// LS Electric XG5000 project: T7_ETH_485_20201209_AfterHeat_Edit
// PLC NewPLC
// module base 0 slot 1: 내장위치결정:XBF-PO02E (오픈컬렉터형, 2축)
// module base 0 slot 2: Cnet:XBL-C41A (Cnet 통신 모듈(RS-422/485))

PROGRAM 7k_pwm (task: 스캔 프로그램)

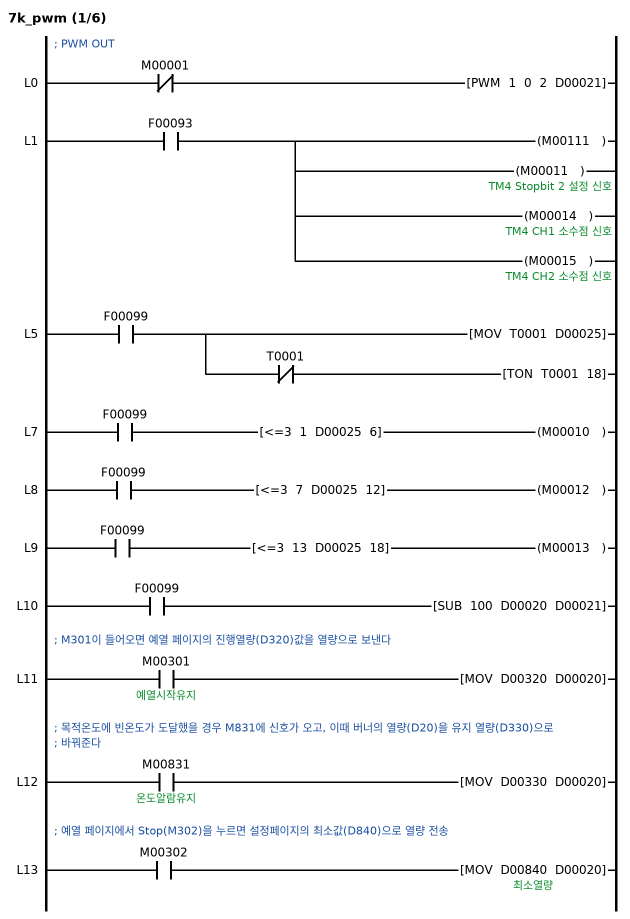
; L0
LOAD NOT  M00001
PWM       1 0 2 D00021
// output comment: PWM OUT
; L1
LOAD      F00093
OUT       M00111
OUT       M00011	// TM4 Stopbit 2 설정 신호
OUT       M00014	// TM4 CH1 소수점 신호
OUT       M00015	// TM4 CH2 소수점 신호
; L5
LOAD      F00099
MOV       T0001 D00025
AND NOT   T0001
TON       T0001 18
; L7
LOAD      F00099
AND<=3    1 D00025 6
OUT       M00010
; L8
LOAD      F00099
AND<=3    7 D00025 12
OUT       M00012
; L9
LOAD      F00099
AND<=3    13 D00025 18
OUT       M00013
; L10
LOAD      F00099
SUB       100 D00020 D00021
; L11
LOAD      M00301	// 예열시작유지
MOV       D00320 D00020
// output comment: M301이 들어오면 예열 페이지의 진행열량(D320)값을 열량으로 보낸다
; L12
LOAD      M00831	// 온도알람유지
MOV       D00330 D00020
// output comment: 목적온도에 빈온도가 도달했을 경우 M831에 신호가 오고, 이때 버너의 열량(D20)을 유지 열량(D330)으로 바꿔준다
; L13
LOAD      M00302
MOV       D00840 D00020	// 최소열량
// output comment: 예열 페이지에서 Stop(M302)을 누르면 설정페이지의 최소값(D840)으로 열량 전송

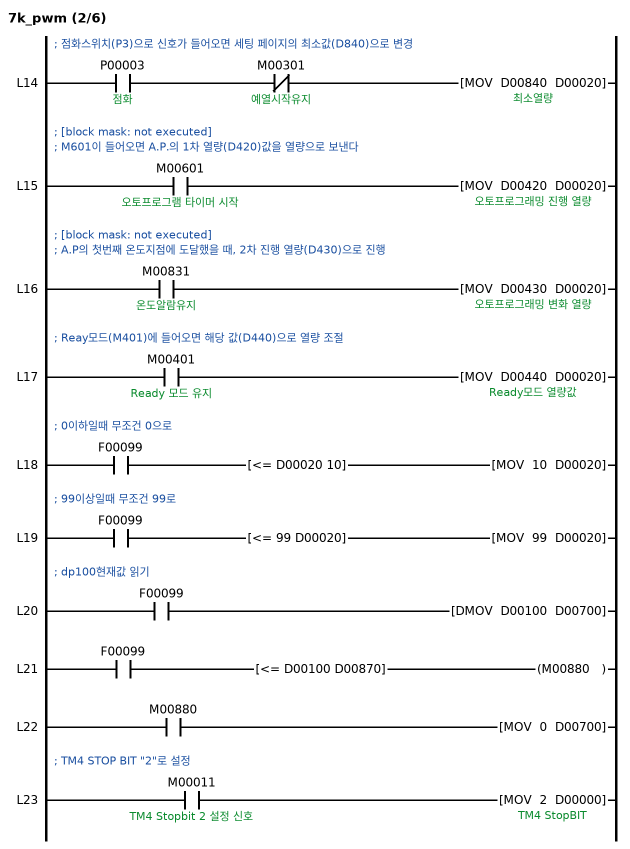
; L14
LOAD      P00003	// 점화
AND NOT   M00301	// 예열시작유지
MOV       D00840 D00020	// 최소열량
// output comment: 점화스위치(P3)으로 신호가 들어오면 세팅 페이지의 최소값(D840)으로 변경
; L15 (block mask: not executed)
LOAD      M00601	// 오토프로그램 타이머 시작
MOV       D00420 D00020	// 오토프로그래밍 진행 열량
// output comment: M601이 들어오면 A.P.의 1차 열량(D420)값을 열량으로 보낸다
; L16 (block mask: not executed)
LOAD      M00831	// 온도알람유지
MOV       D00430 D00020	// 오토프로그래밍 변화 열량
// output comment: A.P의 첫번째 온도지점에 도달했을 때, 2차 진행 열량(D430)으로 진행
; L17
LOAD      M00401	// Ready 모드 유지
MOV       D00440 D00020	// Ready모드 열량값
// output comment: Reay모드(M401)에 들어오면 해당 값(D440)으로 열량 조절
; L18
LOAD      F00099
AND<=     D00020 10
MOV       10 D00020
// output comment: 0이하일때 무조건 0으로
; L19
LOAD      F00099
AND<=     99 D00020
MOV       99 D00020
// output comment: 99이상일때 무조건 99로
; L20
LOAD      F00099
DMOV      D00100 D00700
// output comment: dp100현재값 읽기
; L21
LOAD      F00099
AND<=     D00100 D00870
OUT       M00880
; L22
LOAD      M00880
MOV       0 D00700
; L23
LOAD      M00011	// TM4 Stopbit 2 설정 신호
MOV       2 D00000	// TM4 StopBIT
// output comment: TM4 STOP BIT "2"로 설정

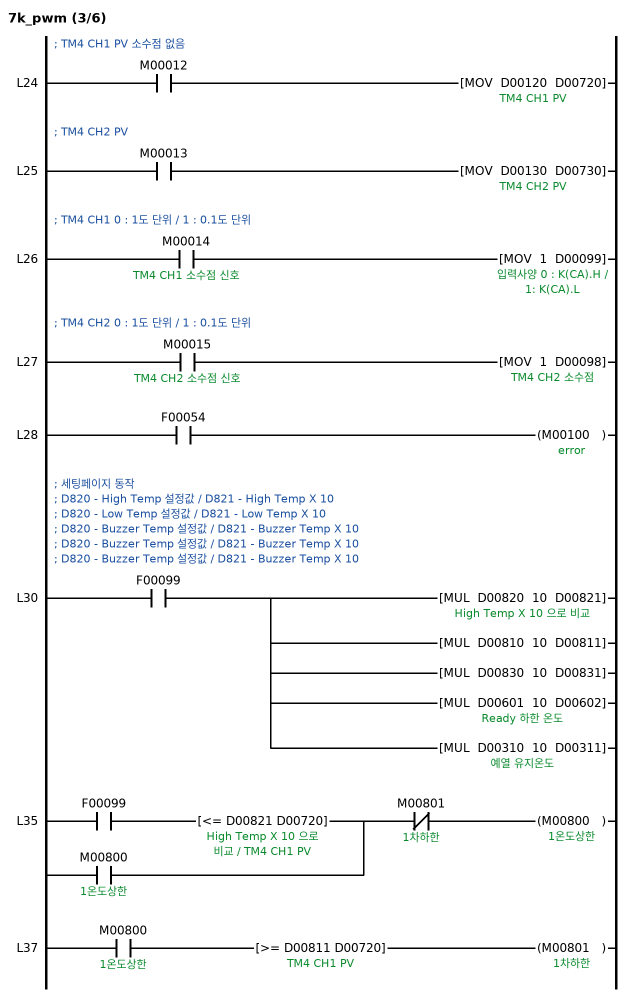
; L24
LOAD      M00012
MOV       D00120 D00720	// TM4 CH1 PV
// output comment: TM4 CH1 PV 소수점 없음
; L25
LOAD      M00013
MOV       D00130 D00730	// TM4 CH2 PV
// output comment: TM4 CH2 PV
; L26
LOAD      M00014	// TM4 CH1 소수점 신호
MOV       1 D00099	// 입력사양 0 : K(CA).H / 1: K(CA).L
// output comment: TM4 CH1 0 : 1도 단위 / 1 : 0.1도 단위
; L27
LOAD      M00015	// TM4 CH2 소수점 신호
MOV       1 D00098	// TM4 CH2 소수점
// output comment: TM4 CH2 0 : 1도 단위 / 1 : 0.1도 단위
; L28
LOAD      F00054
OUT       M00100	// error
// 세팅페이지 동작
; L30
LOAD      F00099
MUL       D00820 10 D00821	// High Temp X 10 으로 비교
MUL       D00810 10 D00811
MUL       D00830 10 D00831
MUL       D00601 10 D00602	// Ready 하한 온도
MUL       D00310 10 D00311	// 예열 유지온도
// output comment: D820 - High Temp 설정값 / D821 - High Temp X 10
// output comment: D820 - Low Temp 설정값 / D821 - Low Temp X 10
// output comment: D820 - Buzzer Temp 설정값 / D821 - Buzzer Temp X 10
// output comment: D820 - Buzzer Temp 설정값 / D821 - Buzzer Temp X 10
// output comment: D820 - Buzzer Temp 설정값 / D821 - Buzzer Temp X 10
; L35
LOAD      F00099
AND<=     D00821 D00720	// High Temp X 10 으로 비교 / TM4 CH1 PV
OR        M00800	// 1온도상한
AND NOT   M00801	// 1차하한
OUT       M00800	// 1온도상한
; L37
LOAD      M00800	// 1온도상한
AND>=     D00811 D00720	// TM4 CH1 PV
OUT       M00801	// 1차하한

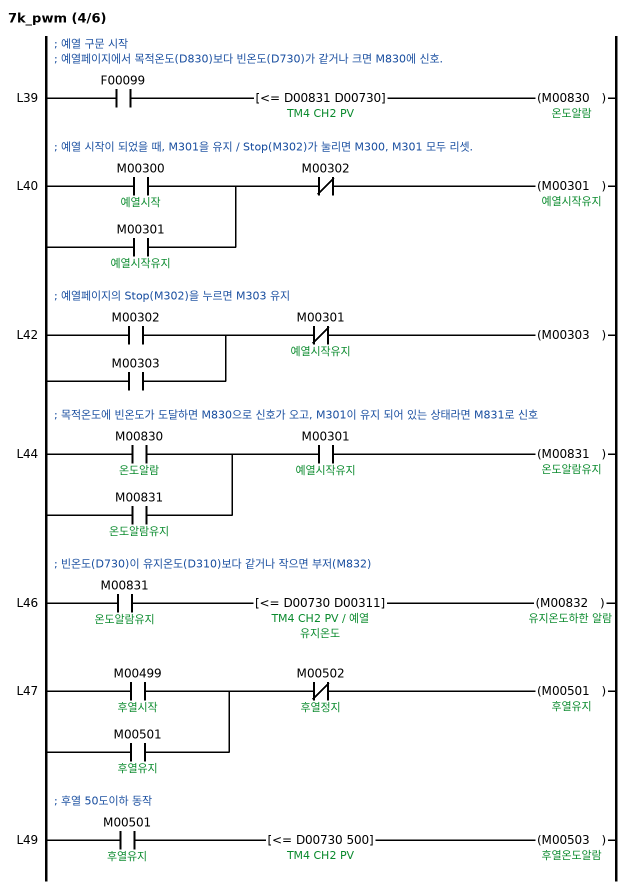
// 예열 구문 시작
; L39
LOAD      F00099
AND<=     D00831 D00730	// TM4 CH2 PV
OUT       M00830	// 온도알람
// output comment: 예열페이지에서 목적온도(D830)보다 빈온도(D730)가 같거나 크면 M830에 신호.
; L40
LOAD      M00300	// 예열시작
OR        M00301	// 예열시작유지
AND NOT   M00302
OUT       M00301	// 예열시작유지
// output comment: 예열 시작이 되었을 때, M301을 유지 / Stop(M302)가 눌리면 M300, M301 모두 리셋.
; L42
LOAD      M00302
OR        M00303
AND NOT   M00301	// 예열시작유지
OUT       M00303
// output comment: 예열페이지의 Stop(M302)을 누르면 M303 유지
; L44
LOAD      M00830	// 온도알람
OR        M00831	// 온도알람유지
AND       M00301	// 예열시작유지
OUT       M00831	// 온도알람유지
// output comment: 목적온도에 빈온도가 도달하면 M830으로 신호가 오고, M301이 유지 되어 있는 상태라면 M831로 신호
; L46
LOAD      M00831	// 온도알람유지
AND<=     D00730 D00311	// TM4 CH2 PV / 예열 유지온도
OUT       M00832	// 유지온도하한 알람
// output comment: 빈온도(D730)이 유지온도(D310)보다 같거나 작으면 부저(M832)
; L47
LOAD      M00499	// 후열시작
OR        M00501	// 후열유지
AND NOT   M00502	// 후열정지
OUT       M00501	// 후열유지
; L49
LOAD      M00501	// 후열유지
AND<=     D00730 500	// TM4 CH2 PV
OUT       M00503	// 후열온도알람
// output comment: 후열 50도이하 동작

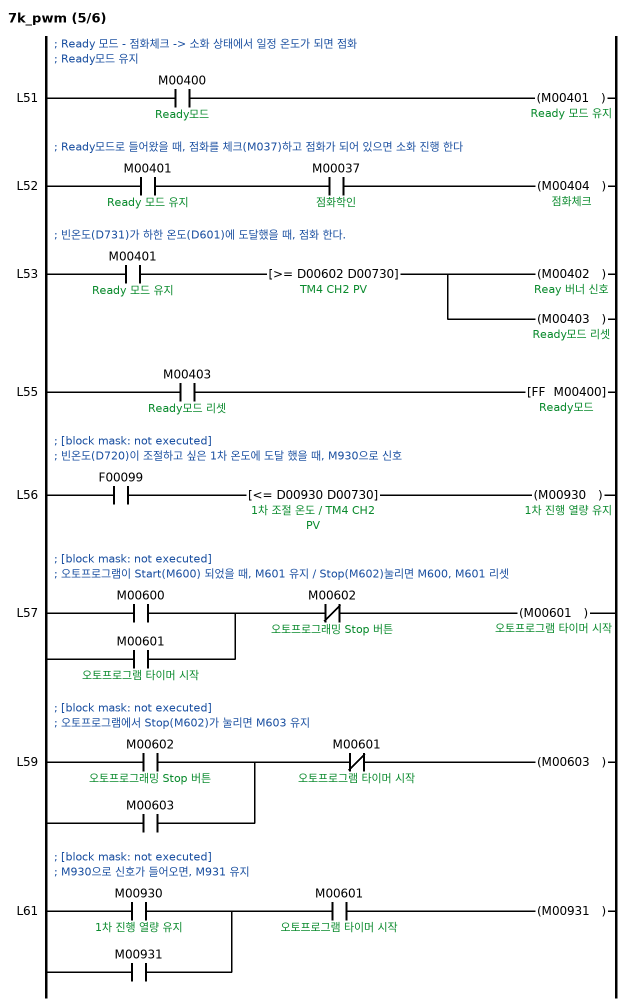
// Ready 모드 - 점화체크 -> 소화 상태에서 일정 온도가 되면 점화
; L51
LOAD      M00400	// Ready모드
OUT       M00401	// Ready 모드 유지
// output comment: Ready모드 유지
; L52
LOAD      M00401	// Ready 모드 유지
AND       M00037	// 점화학인
OUT       M00404	// 점화체크
// output comment: Ready모드로 들어왔을 때, 점화를 체크(M037)하고 점화가 되어 있으면 소화 진행 한다
; L53
LOAD      M00401	// Ready 모드 유지
AND>=     D00602 D00730	// TM4 CH2 PV
OUT       M00402	// Reay 버너 신호
OUT       M00403	// Ready모드 리셋
// output comment: 빈온도(D731)가 하한 온도(D601)에 도달했을 때, 점화 한다.
; L55
LOAD      M00403	// Ready모드 리셋
FF        M00400	// Ready모드
; L56 (block mask: not executed)
LOAD      F00099
AND<=     D00930 D00730	// 1차 조절 온도 / TM4 CH2 PV
OUT       M00930	// 1차 진행 열량 유지
// output comment: 빈온도(D720)이 조절하고 싶은 1차 온도에 도달 했을 때, M930으로 신호
; L57 (block mask: not executed)
LOAD      M00600
OR        M00601	// 오토프로그램 타이머 시작
AND NOT   M00602	// 오토프로그래밍 Stop 버튼
OUT       M00601	// 오토프로그램 타이머 시작
// output comment: 오토프로그램이 Start(M600) 되었을 때, M601 유지 / Stop(M602)눌리면 M600, M601 리셋
; L59 (block mask: not executed)
LOAD      M00602	// 오토프로그래밍 Stop 버튼
OR        M00603
AND NOT   M00601	// 오토프로그램 타이머 시작
OUT       M00603
// output comment: 오토프로그램에서 Stop(M602)가 눌리면 M603 유지
; L61 (block mask: not executed)
LOAD      M00930	// 1차 진행 열량 유지
OR        M00931
AND       M00601	// 오토프로그램 타이머 시작
OUT       M00931
// output comment: M930으로 신호가 들어오면, M931 유지

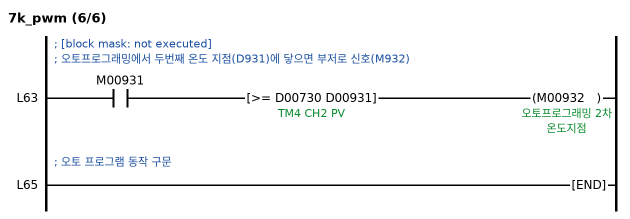
; L63 (block mask: not executed)
LOAD      M00931
AND>=     D00730 D00931	// TM4 CH2 PV
OUT       M00932	// 오토프로그래밍 2차 온도지점
// output comment: 오토프로그래밍에서 두번째 온도 지점(D931)에 닿으면 부저로 신호(M932)
// 오토 프로그램 동작 구문
; L65
END

PROGRAM 타이머 (task: 스캔 프로그램)

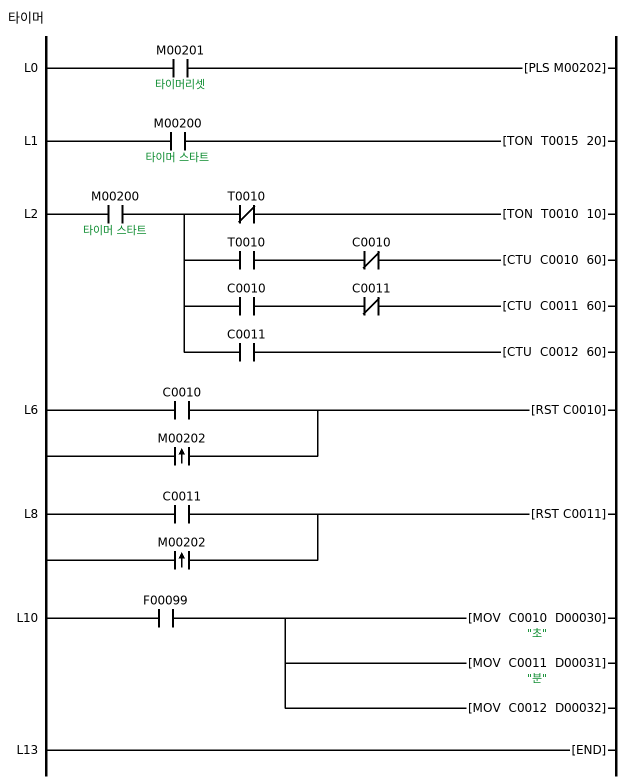
; L0
LOAD      M00201	// 타이머리셋
OUTP      M00202
; L1
LOAD      M00200	// 타이머 스타트
TON       T0015 20
; L2
LOAD      M00200	// 타이머 스타트
MPUSH
AND NOT   T0010
TON       T0010 10
MLOAD
AND       T0010
AND NOT   C0010
CTU       C0010 60
MLOAD
AND       C0010
AND NOT   C0011
CTU       C0011 60
MPOP
AND       C0011
CTU       C0012 60
; L6
LOAD      C0010
ORP       M00202
RST       C0010
; L8
LOAD      C0011
ORP       M00202
RST       C0011
; L10
LOAD      F00099
MOV       C0010 D00030	// "초"
MOV       C0011 D00031	// "분"
MOV       C0012 D00032
; L13
END

PROGRAM control (task: 스캔 프로그램)

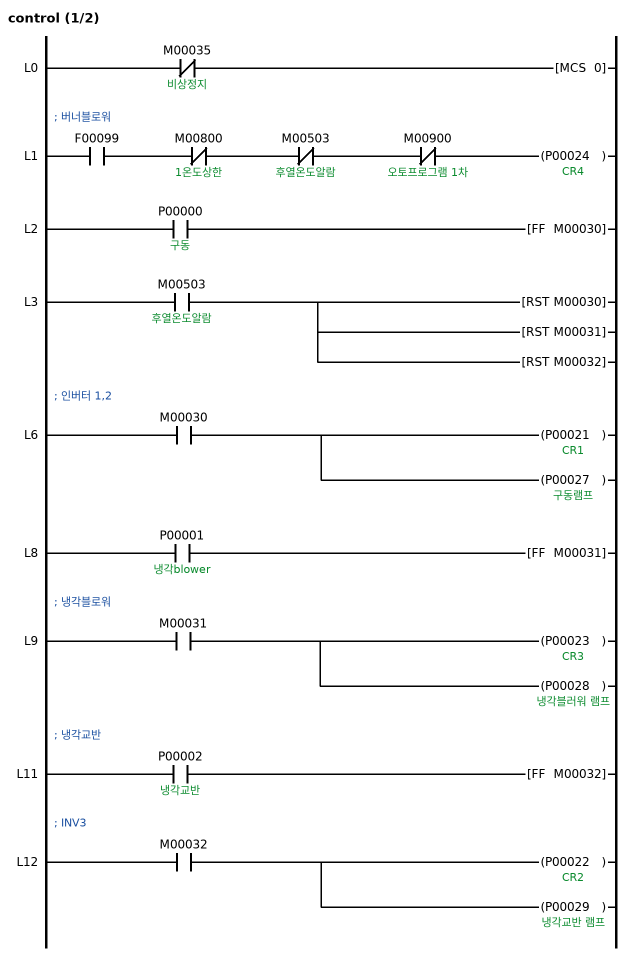
; L0
LOAD NOT  M00035	// 비상정지
MCS       0
; L1
LOAD      F00099
AND NOT   M00800	// 1온도상한
AND NOT   M00503	// 후열온도알람
AND NOT   M00900	// 오토프로그램 1차
OUT       P00024	// CR4
// output comment: 버너블로워
; L2
LOAD      P00000	// 구동
FF        M00030
; L3
LOAD      M00503	// 후열온도알람
RST       M00030
RST       M00031
RST       M00032
; L6
LOAD      M00030
OUT       P00021	// CR1
OUT       P00027	// 구동램프
// output comment: 인버터 1,2
; L8
LOAD      P00001	// 냉각blower
FF        M00031
; L9
LOAD      M00031
OUT       P00023	// CR3
OUT       P00028	// 냉각블러워 램프
// output comment: 냉각블로워
; L11
LOAD      P00002	// 냉각교반
FF        M00032
// output comment: 냉각교반
; L12
LOAD      M00032
OUT       P00022	// CR2
OUT       P00029	// 냉각교반 램프
// output comment: INV3

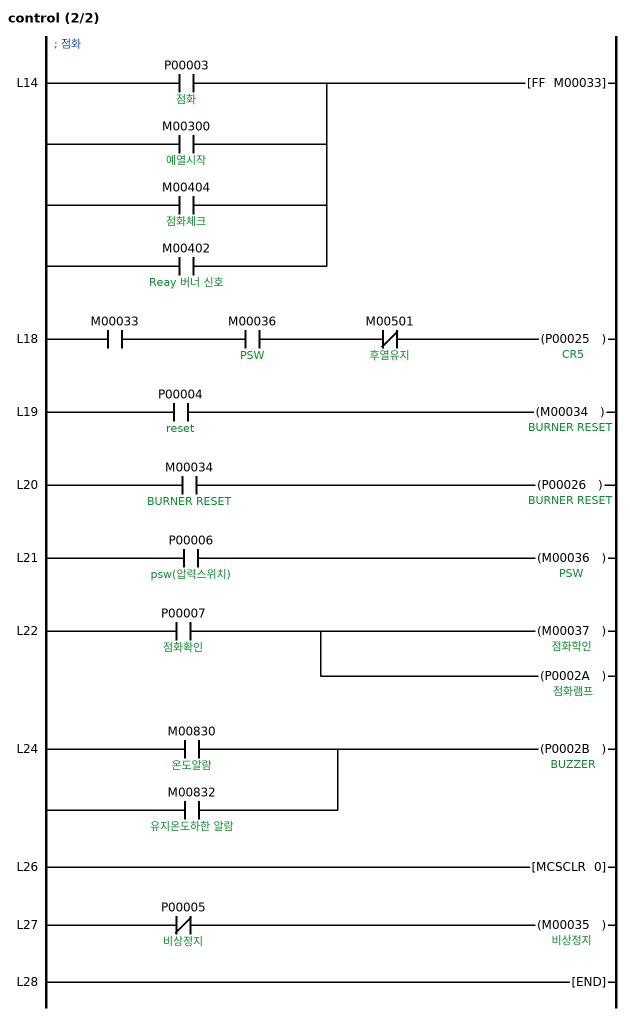
; L14
LOAD      P00003	// 점화
OR        M00300	// 예열시작
OR        M00404	// 점화체크
OR        M00402	// Reay 버너 신호
FF        M00033
// output comment: 점화
; L18
LOAD      M00033
AND       M00036	// PSW
AND NOT   M00501	// 후열유지
OUT       P00025	// CR5
; L19
LOAD      P00004	// reset
OUT       M00034	// BURNER RESET
; L20
LOAD      M00034	// BURNER RESET
OUT       P00026	// BURNER RESET
; L21
LOAD      P00006	// psw(압력스위치)
OUT       M00036	// PSW
; L22
LOAD      P00007	// 점화확인
OUT       M00037	// 점화학인
OUT       P0002A	// 점화램프
; L24
LOAD      M00830	// 온도알람
OR        M00832	// 유지온도하한 알람
OUT       P0002B	// BUZZER
; L26
MCSCLR    0
; L27
LOAD NOT  P00005	// 비상정지
OUT       M00035	// 비상정지
; L28
END

PROGRAM 예열_후열_타이머 (task: 스캔 프로그램)

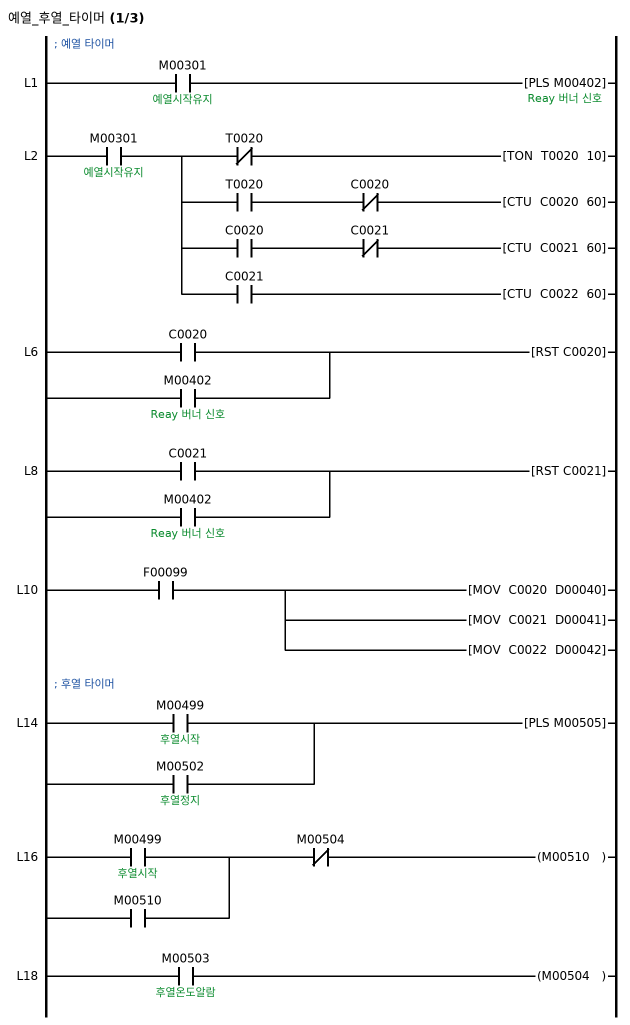
// 예열 타이머
; L1
LOAD      M00301	// 예열시작유지
OUTP      M00402	// Reay 버너 신호
; L2
LOAD      M00301	// 예열시작유지
MPUSH
AND NOT   T0020
TON       T0020 10
MLOAD
AND       T0020
AND NOT   C0020
CTU       C0020 60
MLOAD
AND       C0020
AND NOT   C0021
CTU       C0021 60
MPOP
AND       C0021
CTU       C0022 60
; L6
LOAD      C0020
OR        M00402	// Reay 버너 신호
RST       C0020
; L8
LOAD      C0021
OR        M00402	// Reay 버너 신호
RST       C0021
; L10
LOAD      F00099
MOV       C0020 D00040
MOV       C0021 D00041
MOV       C0022 D00042
// 후열 타이머
; L14
LOAD      M00499	// 후열시작
OR        M00502	// 후열정지
OUTP      M00505
; L16
LOAD      M00499	// 후열시작
OR        M00510
AND NOT   M00504
OUT       M00510
; L18
LOAD      M00503	// 후열온도알람
OUT       M00504

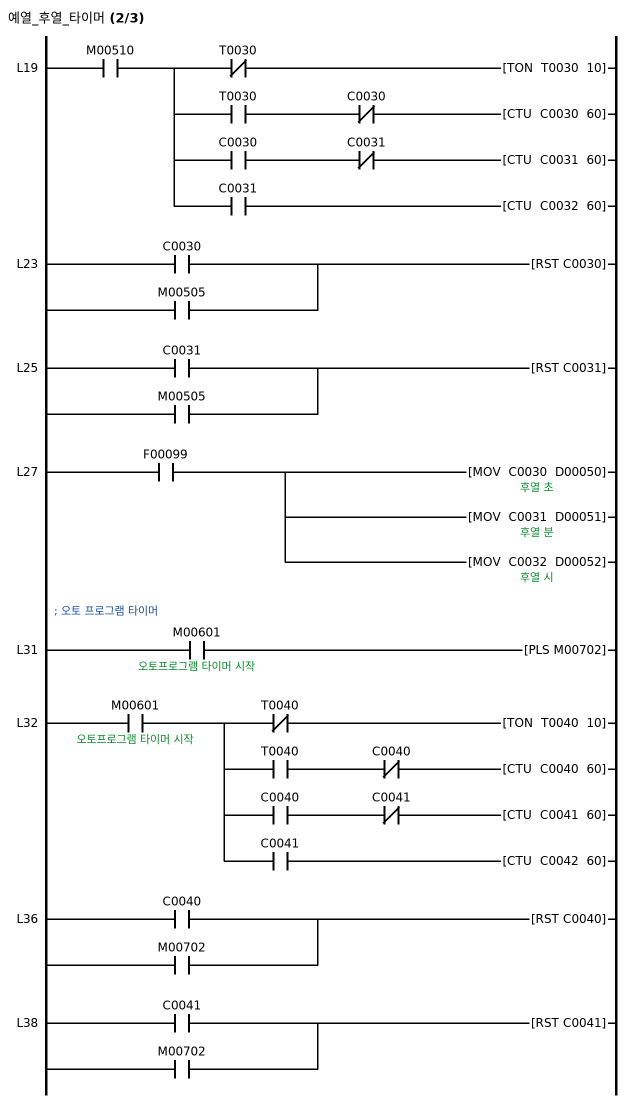
; L19
LOAD      M00510
MPUSH
AND NOT   T0030
TON       T0030 10
MLOAD
AND       T0030
AND NOT   C0030
CTU       C0030 60
MLOAD
AND       C0030
AND NOT   C0031
CTU       C0031 60
MPOP
AND       C0031
CTU       C0032 60
; L23
LOAD      C0030
OR        M00505
RST       C0030
; L25
LOAD      C0031
OR        M00505
RST       C0031
; L27
LOAD      F00099
MOV       C0030 D00050	// 후열 초
MOV       C0031 D00051	// 후열 분
MOV       C0032 D00052	// 후열 시
// 오토 프로그램 타이머
; L31
LOAD      M00601	// 오토프로그램 타이머 시작
OUTP      M00702
; L32
LOAD      M00601	// 오토프로그램 타이머 시작
MPUSH
AND NOT   T0040
TON       T0040 10
MLOAD
AND       T0040
AND NOT   C0040
CTU       C0040 60
MLOAD
AND       C0040
AND NOT   C0041
CTU       C0041 60
MPOP
AND       C0041
CTU       C0042 60
; L36
LOAD      C0040
OR        M00702
RST       C0040
; L38
LOAD      C0041
OR        M00702
RST       C0041

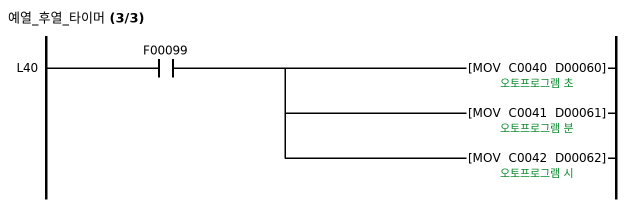
; L40
LOAD      F00099
MOV       C0040 D00060	// 오토프로그램 초
MOV       C0041 D00061	// 오토프로그램 분
MOV       C0042 D00062	// 오토프로그램 시

PROGRAM 485_ARTISAN (task: 스캔 프로그램)

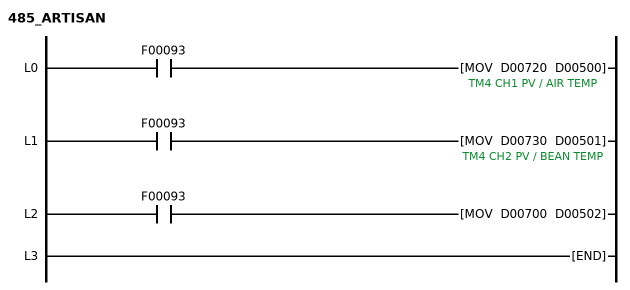
; L0
LOAD      F00093
MOV       D00720 D00500	// TM4 CH1 PV / AIR TEMP
; L1
LOAD      F00093
MOV       D00730 D00501	// TM4 CH2 PV / BEAN TEMP
; L2
LOAD      F00093
MOV       D00700 D00502
; L3
END

VARIABLES AND COMMENTS (devices not used above)
P00020	BIT	BURNER PWM
D00620	WORD	TM4 CH1 PV : 소수점없음
D00600	WORD	Ready Temp